TYPE ST_MappingFileConfig :
STRUCT
	Source : STRING(255);
	Target : STRING(255);
	SourceDataType : E_ConfigDataType;
	TargetDataType : E_ConfigDataType;
	HasTransform : BOOL;
	Scale : LREAL;
	Offset : LREAL;
END_STRUCT
END_TYPE

(* stored: Version 1.1.0.1, ProductVersion 3.1.4026.18
   DUT ST_MappingFileConfig: Id {fbaf5768-c94e-42cf-8a74-7e16c613c462} *)
